PROGRAM ControlFBD
VAR
	qxLampStarted	AT %Q* : BOOL;
	gxSliderAout 	AT %Q* : BOOL; 
	gxSliderAin 	AT %Q* : BOOL; 
	gxSliderBout 	AT %Q* : BOOL; 
	gxSliderBin 	AT %Q* : BOOL; 
	gxDrillDown 	AT %Q* : BOOL;
	gxDrillUp		AT %Q* : BOOL;
	
	ixButtonStart	AT %I* : BOOL;
	ixButtonStop	AT %I* : BOOL;
	ixSliderAout	AT %I* : BOOL;
	ixSliderAin		AT %I* : BOOL;
	ixSliderBout	AT %I* : BOOL;
	ixSliderBin		AT %I* : BOOL;
	ixDrillUp		AT %I* : BOOL;
	ixDrillDown		AT %I* : BOOL;

END_VAR

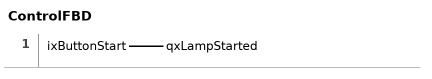
// NETWORK 1
qxLampStarted := ixButtonStart;

END_PROGRAM

(* stored: Version 1.1.0.1, ProductVersion 3.1.4024.11
   POU ControlFBD: Id {441bf843-2f16-42db-a10b-d561aec11b1f}, SpecialFunc None *)
